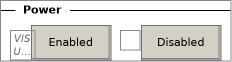
VISUALIZATION VISU_BaseAxis_Power  // 232x62
VAR_IN_OUT
	axis : BaseAxis;
    axisWidget : BaseAxisWidget;
END_VAR
    Button (141,25 80x35), "Disabled", input disabled if: axis.processes.power.statuses.enabledStatus.disabled
        OnMouseClick: execute { axis.processes.power.set.enable := FALSE; axis.processes.power.do_request := TRUE; }
    Frame (120,30 20x20)
        shows VISU_State_gray_orange(state := axis.statuses.poweredStatus.disabled)
    Button (31,25 80x35), "Enabled", input disabled if: axis.processes.power.statuses.enabledStatus.disabled
        OnMouseClick: execute { axis.processes.power.set.enable := TRUE; axis.processes.power.do_request := TRUE; }
    Frame (10,30 25x30)
        shows VISU_State_gray_green(state := axis.statuses.poweredStatus.enabled)
    Label (20,0 55x20), "Power"
    Line (70,10) (230,10)
    Line (0,10) (15,10)
END_VISUALIZATION

(* stored: Version 1.1.0.1, ProductVersion 3.1.4019.2
   Visu VISU_BaseAxis_Power: Id {22b512da-57a5-4a32-8339-f2c88fa1eaaf} *)
